// TIA Portal V19 export
TYPE "C301_VAR_VEN_TYPIC"
   STRUCT
      STS { ExternalAccessible := 'False'; ExternalVisible := 'False'; ExternalWritable := 'False'} : USInt;   // Status van de ventilator
      DIR { ExternalAccessible := 'False'; ExternalVisible := 'False'; ExternalWritable := 'False'} : USInt;   // Richting van de ventilator
      BMO { ExternalAccessible := 'False'; ExternalVisible := 'False'; ExternalWritable := 'False'} : USInt;   // Bedieningsmode
      BST { ExternalAccessible := 'False'; ExternalVisible := 'False'; ExternalWritable := 'False'} : USInt;   // Bestuurbaarheid
      PWR { ExternalAccessible := 'False'; ExternalVisible := 'False'; ExternalWritable := 'False'} : Real;   // Vermogen van de ventilator
      TYD_TOT_AAN { ExternalAccessible := 'False'; ExternalVisible := 'False'; ExternalWritable := 'False'} : USInt;   // Totaal aantal draaiuren
   END_STRUCT;
END_TYPE
